(* PLC project LPC POUs, Beremiz Beremiz 0.0 *)
(* stored: creationDateTime 2008-12-14T16:53:26, modificationDateTime 2012-01-20T13:35:46 *)

FUNCTION_BLOCK DEW_POINT
  VAR_INPUT
    RH : REAL;
    TEMP : REAL;
  END_VAR
  VAR_OUTPUT
    DEW_POINT : REAL;
  END_VAR

		if RH < 0.0 then
		  RH := 0.0;
		end_if;
		if RH > 100.0 then
		  RH := 100.0;
		end_if;
		DEW_POINT:=sqrt(sqrt(sqrt(RH/100.0)))*(112.0+(0.9*TEMP))+(0.1*TEMP)-112.0;
			
END_FUNCTION_BLOCK

FUNCTION_BLOCK GET_RETAIN_DATA
  VAR_INPUT
    INDEX : UINT := 0;  (* Index (row) of the retain array. *)
    READ : BOOL := FALSE;
  END_VAR
  VAR_OUTPUT
    WORD1 : UINT;  (* Data - first column. *)
    WORD2 : UINT;
    WORD3 : UINT;
    RD_OK : BOOL := FALSE;
  END_VAR

{
extern IEC_UINT __GetRetainData(BOOL, IEC_UINT, IEC_UINT);
extern BOOL __GetReadStatus(BOOL);
__SET_VAR(data__->,WORD1,__GetRetainData(__GET_VAR(data__->READ),__GET_VAR(data__->INDEX),0));
__SET_VAR(data__->,WORD2,__GetRetainData(__GET_VAR(data__->READ),__GET_VAR(data__->INDEX),1));
__SET_VAR(data__->,WORD3,__GetRetainData(__GET_VAR(data__->READ),__GET_VAR(data__->INDEX),2));
__SET_VAR(data__->,RD_OK,__GetReadStatus(0));
}
          
END_FUNCTION_BLOCK

FUNCTION_BLOCK SET_RETAIN_DATA
  VAR_INPUT
    INDEX : UINT := 0;
    WRITE : BOOL := FALSE;
    WORD1 : UINT;
    WORD2 : UINT;
    WORD3 : UINT;
  END_VAR
  VAR_OUTPUT
    WR_OK : BOOL := FALSE;
  END_VAR

{
extern BOOL __SetRetainData(BOOL, IEC_UINT, IEC_UINT, IEC_UINT, IEC_UINT);
__SET_VAR(data__->,WR_OK,__SetRetainData(__GET_VAR(data__->WRITE),__GET_VAR(data__->INDEX),__GET_VAR(data__->WORD1),__GET_VAR(data__->WORD2),__GET_VAR(data__->WORD3)));
}
          
END_FUNCTION_BLOCK

FUNCTION_BLOCK FIND_RETAIN_DATA
  VAR_OUTPUT
    FOUND : BOOL := False;
    INDEX : UINT;
  END_VAR
  VAR_INPUT
    START_IDX : UINT := 0;
    END_IDX : UINT := 0;
    SEARCH : BOOL := False;
    WORD1 : UINT;
    WORD2 : UINT;
    WORD3 : UINT;
  END_VAR

{
extern BOOL __FindRetainData(BOOL, IEC_UINT, IEC_UINT, IEC_UINT, IEC_UINT, IEC_UINT);
extern IEC_UINT __GetFoundIndex(BOOL);
__SET_VAR(data__->,FOUND,__FindRetainData(__GET_VAR(data__->SEARCH),__GET_VAR(data__->START_IDX),__GET_VAR(data__->END_IDX),__GET_VAR(data__->WORD1),__GET_VAR(data__->WORD2),__GET_VAR(data__->WORD3)));
__SET_VAR(data__->,INDEX,__GetFoundIndex(0));
}
          
END_FUNCTION_BLOCK

FUNCTION_BLOCK PID_A
  VAR_INPUT
    SET_POINT : REAL;
  END_VAR
  VAR
    ena : INT := 1;
  END_VAR
  VAR_INPUT
    ACTUAL_VALUE : REAL;
    REVERSE : BOOL;
    HOLD : BOOL;
    MANUAL : BOOL;
    MANUAL_REF : REAL;
    Kp_GAIN : REAL;
    Ki_GAIN : REAL;
    Kd_GAIN : REAL;
    Td_FADEOUT : TIME := t#1s;
    DEAD_BAND : REAL;
    OUT_MAX : REAL;
    OUT_MIN : REAL;
    CYCLE_TIME : TIME := t#0.1s;
  END_VAR
  VAR_OUTPUT
    OUT : REAL;
  END_VAR
  VAR
    D_fadeout : REAL;
    Error_n : REAL := 0.0;
    Error_n1 : REAL := 0.0;
    Error_n2 : REAL := 0.0;
    Dout_n : REAL := 0.0;
    Dout : REAL := 0.0;
    Dout_1 : REAL := 0.0;
    TON_1 : TON;
    TON_1_Q : BOOL;
    ET1 : TIME;
    CTr : REAL;
    FTr : REAL;
    power : REAL;
    OUTchk : REAL;
    Dout_int : REAL;
    Reverse_1 : BOOL;
    Soft_t : BOOL;
    R_chk : INT;
  END_VAR

TON_1(
     IN := NOT TON_1_Q,
     PT := CYCLE_TIME,
     Q => TON_1_Q,
     ET => ET1
     );
if TON_1_Q then
  if REVERSE then
    Error_n := SET_POINT - ACTUAL_VALUE;
  else
    Error_n := ACTUAL_VALUE - SET_POINT;
  end_if;
  if Td_FADEOUT <= T#0.05s then
  Td_FADEOUT := t#0.05s;
  end_if;
     CTr := TIME_TO_REAL (CYCLE_TIME);
     FTr := TIME_TO_REAL (Td_FADEOUT);
      power := CTr / FTr;
       D_Fadeout := EXPT( 0.04979 , power );  (*time to reach 5% = e^(-3) *)
         Dout := Kd_GAIN * (Error_n - 2.0 * Error_n1 + Error_n2); 
         Dout_n := Dout + Dout_1 * D_Fadeout;  
         Dout_int := Dout_int + Dout_n;
           OUTchk := OUTchk + Kp_GAIN * (Error_n - Error_n1) + Ki_GAIN * Error_n * CTr;
    R_chk:= bool_to_int(REVERSE) + bool_to_int(Reverse_1);
        if (Soft_t or R_chk=1) then
         Dout_int := 0.0;
          Dout_n := 0.0;
           Dout_1:= 0.0;
            Dout:= 0.0;
            OUTchk:= OUT;
           Error_n1:=Error_n;
          Error_n2:=Error_n;
         Soft_t := 0;
        end_if;
      if R_chk =1 then 
        Error_n:=0.0;
        Soft_t := True;
      end_if;
           
     if OUTchk > OUT_MAX then
        OUTchk := OUT_MAX;
     end_if;
     
     if OUTchk < OUT_MIN then
        OUTchk := OUT_MIN;
     end_if;
    
  if MANUAL then
    OUT := MANUAL_REF;
     OUTchk:= OUT;
      Dout_int := 0.0;
       Dout_n := 0.0;
       Dout_1:= 0.0;
  else 
    if abs(Error_n) < DEAD_BAND or HOLD  then
       OUT := OUT;
        OUTchk:= OUT;
        Dout_int := 0.0;
        Dout_n := 0.0;
       Dout_1:= 0.0;
    else
      OUT := OUTchk + Dout_int;
    end_if;
  end_if;
  
 if OUT > OUT_MAX then
 OUT := OUT_MAX;
 end_if;
  
 if OUT < OUT_MIN then
 OUT := OUT_MIN;
 end_if;
 
    Error_n2 := Error_n1;
     Error_n1 := Error_n;
      Dout_1:=Dout_n;
        Reverse_1 := REVERSE;
else
  OUT:=OUT;
end_if;
          
END_FUNCTION_BLOCK
